FUNCTION_BLOCK F_LOWER_BOUND (* Returns the lower bound of the dimension of the given array *)
  (* Standard: 61131-3; Description: Copyright (c) 2026 Demmler Andreas Fahrzeugbau This program and the accompanying materials are made available under the terms of the Eclipse Public License 2.0 which is available at https://www.eclipse.org/legal/epl-2.0/ SPDX-License-Identifier: EPL-2.0 *)
  (* Version 1.0, 2026-01-23, Franz H??pfinger, Demmler Andreas Fahrzeugbau, Initial Implementation *)
  PACKAGE iec61131::arrays;
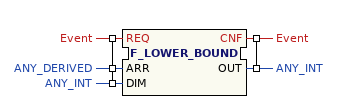
  EVENT_INPUT
    REQ WITH ARR, DIM; (* Service Request *)
  END_EVENT
  EVENT_OUTPUT
    CNF WITH OUT; (* Confirmation of Requested Service *)
  END_EVENT
  VAR_INPUT
    ARR : ANY_DERIVED; (* input array *)
    DIM : ANY_INT := UDINT#1; (* Dimension, 1-based *)
  END_VAR
  VAR_OUTPUT
    OUT : ANY_INT; (* lowest index of the Dimension *)
  END_VAR
  EC_STATES
    REQ : REQ -> CNF;
  END_STATES
  ALGORITHM REQ IN ST:
OUT := LOWER_BOUND(ARR, DIM);
  END_ALGORITHM
END_FUNCTION_BLOCK
